// TIA Portal V16 export
// export: Created 2023-08-28T09:37:54.1315552Z, ExportSetting WithDefaults, DisplayName Totally Integrated Automation Portal, DisplayVersion V16 Update 6, DisplayName TIA Portal Version Control Interface, DisplayVersion V16 Update 2, DisplayName TIA Portal Openness, DisplayVersion V16 Update 6, DisplayName STEP 7 Professional, DisplayVersion V16 Update 6, DisplayName STEP 7 Safety, DisplayVersion V16, DisplayName WinCC Advanced, DisplayVersion V16 Update 6
VAR_GLOBAL   // PLC tag table "RTC"
   status_rd_sys_t AT %MW200 : Int;
   status_rd_loc_t AT %MW202 : Int;
   Ustaw_czas AT %M206.0 : Bool;
   trig_ustaw_czas AT %M206.1 : Bool;
   status_wr_sys_t AT %MW204 : Int;
   trig_pobierz_czas AT %M206.3 : Bool;
   Pobierz_czas AT %M206.2 : Bool;
END_VAR
